FUNCTION_BLOCK FB_MovingAverageReal
VAR_INPUT
	ValueToAdd : LREAL;
END_VAR
VAR_IN_OUT
	AverageArray  : ARRAY [*] OF LREAL;
END_VAR
VAR_OUTPUT
	CurrentValue : LREAL;
END_VAR
VAR
	CurrentIndex : UINT;
	NumValues: UINT;
END_VAR
VAR_TEMP
	I: DINT;
	Sum: LREAL;
	ArrayLength : UINT;
END_VAR

// Compute average over array.
// The order of this addition and MOD are important to avoid going out of bounds.
// NOTE: We deliberately do not try to account for underfilling the array.
ArrayLength := TO_UINT(UPPER_BOUND(AverageArray, 1) - LOWER_BOUND(AverageArray, 1) + 1);
AverageArray[CurrentIndex] := ValueToAdd;
CurrentIndex := CurrentIndex + 1;
CurrentIndex := CurrentIndex MOD ArrayLength;
NumValues := MIN(NumValues + 1 , ArrayLength);
// This wastes a little time walking pointless values if the array is underfilled,
// but they are zero initialized and thus should not afffect the calculation.
FOR I := LOWER_BOUND(AverageArray, 1) TO UPPER_BOUND(AverageArray, 1) BY 1 DO
	Sum := Sum + AverageArray[I];
END_FOR
CurrentValue := TO_REAL(Sum / NumValues);

END_FUNCTION_BLOCK

(* stored: Version 1.1.0.1, ProductVersion 3.1.4022.16
   POU FB_MovingAverageReal: Id {fda7e211-5c6c-492f-ac36-81cea3ee5c49}, SpecialFunc None *)
